TYPE U_CNC_Fanuc_Input :
UNION
	aStdIn		AT %I*		:ARRAY [1..32] OF UINT;
	Status					:ST_CNC_Robot_Status;	
END_UNION
END_TYPE

(* stored: Version 1.1.0.1, ProductVersion 3.1.4024.12
   DUT U_CNC_Fanuc_Input: Id {632e8594-ac45-4067-a795-d3411a6c9602} *)
